(*
SPDX-FileCopyrightText: © 2026 Oleksandr Tiutyk <trofimich@gmail.com>
SPDX-License-Identifier: MIT
License: https://opensource.org/license/mit
*)

(*!
<summary>Enumerates the current storage slots of a Dictionary.</summary>
<description>
The source is borrowed and must outlive the cursor. Enumeration has no guaranteed ordering. Do not mutate the
source during traversal. Current is a borrowed view and must not be released or modified as an owning
descriptor; it is invalidated by cursor advancement/reset or source mutation. The caller owns and explicitly
releases a dynamically created cursor. MoveNext stops advancing at the end position of an unchanged source;
repeated exhausted calls return FALSE until Reset.
A null constructor source is diagnosed by traversal/current access, never by FB_init.
</description>
*)

{attribute 'no_explicit_call' := 'do not call this function block directly'}
{attribute 'enable_dynamic_creation'}
FUNCTION_BLOCK DictionaryEnumerator EXTENDS TOF_Core.Object IMPLEMENTS TOF_Core.IEnumerator
VAR_STAT
	//! <summary>Class name shared by all instances of this function block.</summary>
	{attribute 'hide'} 
	_ClassName : STRING := __POUNAME();
END_VAR
VAR
	{attribute 'hide'} 
	_Dictionary : IReadOnlyDictionary;
	{attribute 'hide'} 
	_CurrentIndex : DINT := -1;
	
	{attribute 'hide'} 
	_GenericKeyValuePair : TOF_Core.GENERIC_KEY_VALUE_PAIR;
	{attribute 'hide'} 
	_GenericValue : TOF_Core.GENERIC_VALUE;	
END_VAR

(*!
<summary>Borrows the concrete cursor class name without transferring storage ownership.</summary>
*)
{attribute 'monitoring' := 'call'}
PROPERTY ClassName : REFERENCE TO STRING
GET
ClassName REF= _ClassName;
END_GET
END_PROPERTY

(*!
<summary>Exposes a read-only borrowed view of the current entry.</summary>
<description>
Reading Current before the first successful MoveNext, after Reset or after exhaustion yields an empty
descriptor. Otherwise payload is borrowed, with no disposal rights. Do not modify or release the descriptor.
The view may change on subsequent property access, cursor movement or source mutation. The outer USER_DEFINED
value points to cursor-local GENERIC_KEY_VALUE_PAIR storage; nested descriptors borrow collection payload.
Missing source raises DataMemberNotSpecifiedException before source access or cursor advancement.
</description>
*)
{attribute 'monitoring' := 'call'}
PROPERTY FINAL Current : REFERENCE TO TOF_Core.GENERIC_VALUE
GET
requireSource();

IF _CurrentIndex >= 0 AND_THEN _CurrentIndex < _Dictionary.Length THEN
	_GenericKeyValuePair := _Dictionary.GetKeyValuePairByIndex(index := _CurrentIndex); 
	_GenericValue := TOF_Core.GenericValueFactory.FromParts(
		genericTypeClass := TOF_Core.GENERIC_TYPE_CLASS.USER_DEFINED,
		address := ADR(_GenericKeyValuePair),
		size := SIZEOF(TOF_Core.GENERIC_KEY_VALUE_PAIR),
		memoryManagementBehavior := TOF_Core.GENERIC_MEMORY_MANAGEMENT_BEHAVIOR.STORE_ORIGINAL_REFERENCE_AND_NOT_OWNS_MEMORY
	);
ELSE
	_GenericValue.Reset();
END_IF 

Current REF= _GenericValue;
END_GET
END_PROPERTY

(*!
<summary>Returns the current entry in its concrete representation.</summary>
<description>
Use only after MoveNext returns TRUE and before the next cursor or source change. No result is promised
outside a valid position. Nested descriptors borrow payload; their owner flags do not transfer disposal
rights.
Missing source raises DataMemberNotSpecifiedException before source access or cursor advancement.
</description>
*)
PROPERTY FINAL CurrentKeyValuePair : TOF_Core.GENERIC_KEY_VALUE_PAIR
GET
requireSource();

IF _CurrentIndex >= 0 AND_THEN _CurrentIndex < _Dictionary.Length THEN
	CurrentKeyValuePair := _Dictionary.GetKeyValuePairByIndex(index := _CurrentIndex); 
END_IF
END_GET
END_PROPERTY

(*!
<summary>Binds the borrowed source for enumeration.</summary>
<description>
The source must be non-null and outlive the cursor. Only the reference is assigned; no allocation, callbacks
or throwing validation are performed. A null source remains invalid configuration and is reported by
MoveNext or current-value access without throwing from initialization.
</description>
*)
METHOD FB_init : BOOL
VAR_INPUT
	bInitRetains : BOOL; // TRUE: the retain variables are initialized (reset warm / reset cold)
	bInCopyCode : BOOL;  // TRUE: the instance will be copied to the copy code afterward (online change)
	dictionary : IReadOnlyDictionary;
END_VAR
_Dictionary := dictionary;
END_METHOD

(*!
<summary>Advances the cursor to the next source position.</summary>
<description>
The source must be live, non-null and structurally unchanged during traversal. TRUE identifies a current
entry. The index advances only while below source Length and stops at the end position. Repeated exhausted
calls return FALSE without incrementing the index; reading Current yields an empty descriptor. Reset allows
traversal from the beginning again. No snapshot or mutation detection is provided.
Missing source raises DataMemberNotSpecifiedException before source access or cursor advancement.
</description>
*)
{attribute "object_name" := "MoveNext"}
METHOD FINAL MoveNext : BOOL
requireSource();

IF _CurrentIndex < _Dictionary.Length THEN
	_CurrentIndex := _CurrentIndex + 1;
END_IF

MoveNext := _CurrentIndex < _Dictionary.Length;
END_METHOD

(*!
<summary>Provides the library namespace for diagnostics.</summary>
<description>
Borrowed read-only reference to compiler-initialized metadata; no ownership transfer.
</description>
*)
{attribute 'monitoring' := 'call'}
PROPERTY NamespaceName : REFERENCE TO STRING
GET
NamespaceName REF= CurrentNamespace.Name;
END_GET
END_PROPERTY

(*!
<summary>Places the cursor before the first source entry.</summary>
<description>
The next MoveNext starts at zero. Does not modify the source or release payload; reading Current now yields an
empty descriptor. Descendants cannot override this cursor operation; advancement, reset and borrowed current
views use the same cursor state.
</description>
*)
{attribute "object_name" := "Reset"}
METHOD FINAL Reset
_CurrentIndex := -1;
END_METHOD

(*!
<summary>Reports the size of this function-block instance.</summary>
<description>
Measured in bytes; includes inline storage but excludes separately allocated buffers, payload and enumerators.
</description>
*)
{attribute 'monitoring' := 'call'}
PROPERTY SelfSize : ULINT
GET
SelfSize := XSIZEOF(THIS^);
END_GET
END_PROPERTY

(*!
<summary>Requires the configured source before traversal or current-value access.</summary>
<description>
A missing mandatory source is configuration failure, not an empty collection. Raises a framework diagnostic
outside lifecycle methods and before mutation; it does not validate arbitrary pointer lifetime.
</description>
*)
METHOD PRIVATE requireSource
IF _Dictionary = 0 THEN
	TOF_Core.Exceptions.ThrowDataMemberNotSpecified(
		sourceNamespaceName := NamespaceName,
		sourceClassName := ClassName,
		sourcePOUName := __POUNAME(),
		sourcePosition := __POSITION(),
		dataMemberName := 'dictionary'
	);
END_IF
END_METHOD

END_FUNCTION_BLOCK

(* stored: Version 1.1.0.1
   POU DictionaryEnumerator: Id {2f365963-7036-4f79-8584-bc80ea1e769d}, SpecialFunc None
   Property ClassName: Id {839d6121-03b1-4336-9ccf-f78a04cd0cb5}
   Get Get: Id {e0aa9b3a-9a64-4398-b874-5ed4b802f8a8}
   Property Current: Id {9d7a3084-f2d9-46a4-babc-c0d4307e4c92}
   Get Get: Id {f0a9af6e-a818-4733-9637-b26e3a47ceb1}
   Property CurrentKeyValuePair: Id {a11fa9ca-d7fd-47e7-8c94-382211eba30f}
   Get Get: Id {587ce946-29e3-488a-a34c-6505b64fa177}
   Method FB_init: Id {5f1ac79b-7b16-408a-a050-ca6526d9c743}
   Method MoveNext: Id {a3b96f77-158c-4502-97c9-c508c77c0dd2}
   Property NamespaceName: Id {2825246a-435d-4d7f-beb7-b17a1356bf70}
   Get Get: Id {88723d2e-40ed-4daf-8b32-5e90b0fb1460}
   Method Reset: Id {ffc13050-106a-4a43-ad03-55630a53602f}
   Property SelfSize: Id {1db19b22-0572-4a68-948e-fa84d0bb1deb}
   Get Get: Id {ee09e011-6acd-46b1-94f4-d278acd0fb55}
   Method requireSource: Id {ae3d8648-b07a-445a-902c-01ee2ce8366d} *)
